INTERFACE I_PersistentDataStorage

PROPERTY TriggerWriteOfPersistentData : BOOL
GET
END_GET
SET
END_SET
END_PROPERTY

END_INTERFACE

(* stored: Version 1.1.0.1
   Itf I_PersistentDataStorage: Id {ef419ae2-fd84-4184-8b85-555366ae9e1e}
   Property TriggerWriteOfPersistentData: Id {86860e44-3b34-47eb-8399-bfd63ac490b7}
   Get Get: Id {12f351ed-ba76-4162-ae25-4323bca9b375}
   Set Set: Id {ee8dd903-df53-4076-848c-3bbc1f980f73} *)
